Staubli VAL3: N21_Dosi.pgx

program N21_Dosi()
  local pointRx l_pDosi
begin

  // Anar al punt de dosificar placa
  if aioGet(aiNumPipeta)==2
    l_pDosi=pDosi8[aioGet(aiNumPlacaDosi)]
  else
    l_pDosi=pDosi1[aioGet(aiNumPlacaDosi)]
  endIf
  l_pDosi.trsf.x=l_pDosi.trsf.x+nXOffset
  l_pDosi.trsf.y=l_pDosi.trsf.y+nYOffset
  l_pDosi.trsf.z=l_pDosi.trsf.z+nZOffset
  l_pDosi.trsf.rx=l_pDosi.trsf.rx+aioGet(aiAngleInclinarPipieta)

  movel(l_pDosi,tToolActiva,mLent)
  waitEndMove()

  bTaskDone=true
end
